FUNCTION_BLOCK FB_CsvReader
VAR_INPUT
	
END_VAR
VAR_OUTPUT
	data : ARRAY [0..100] OF T_MaxString;
END_VAR

VAR
	sNetId : T_MaxString := '';
	bOpen : BOOL;
	bClose : BOOL;
	
	fbOpen : FB_FileOpen;
	fbGets : FB_FileGets;
	fbClose : FB_FileClose;
	
	n : UDINT;
	i : UDINT;

	
	
	
	eState : UINT;
END_VAR

n := n + 1;
CASE eState OF
	0 : // Idle
		i := 0;
	
	1 : // Start open
		fbOpen(
			sNetId := sNetId,
			sPathName := 'C:\test.txt',
			nMode := FOPEN_MODEREAD OR FOPEN_MODETEXT,
			ePath := PATH_GENERIC,
			bExecute := TRUE
		);
		
		eState := 2;
	
	2 : // Open
		fbOpen(bExecute := FALSE);
		
		IF NOT fbOpen.bBusy AND NOT fbOpen.bError THEN
			eState := 3;
		END_IF
		
	3 : // Ready
		fbGets(
			sNetId := sNetId,
			hFile := fbOpen.hFile,
			bExecute := TRUE
		);
		
		eState := 4;
		
	4 :
		fbGets(bExecute := FALSE);
		
		IF NOT fbGets.bBusy AND NOT fbGets.bError THEN
			IF NOT fbGets.bEOF THEN
				data[i] := CONCAT(UDINT_TO_STRING(n), fbGets.sLine);
				
				i := i + 1;
				eState := 3;
				
			ELSE
				eState := 100;
				
			END_IF
		END_IF
	
	100 : // Start close
		fbClose(
			sNetId := sNetId,
			hFile := fbOpen.hFile,
			bExecute := TRUE
		);
		
		eState := 101;
		
	101: // Close
		fbClose(bExecute := FALSE);
		
		IF NOT fbClose.bBusy AND NOT fbClose.bError THEN
			eState := 0;
			
		END_IF
		
	
END_CASE

END_FUNCTION_BLOCK

(* stored: Version 1.1.0.1, ProductVersion 3.1.4022.18
   POU FB_CsvReader: Id {3731b04a-1903-4e40-9513-292cb4a2684f}, SpecialFunc None *)
